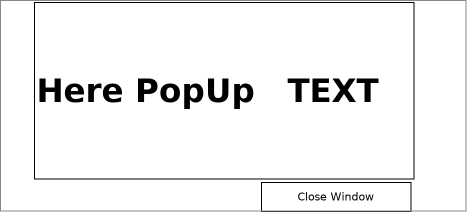
VISUALIZATION W01_PopupScreen  // 467x212
    Label (24,34 443x139)
    RoundedRectangle (261,182 150x30), "Close Window"
        OnMouseClick: CloseDialog Dialog=W01_PopupScreen, Result=OK, NumpadKeypadSet=True
    Rectangle (34,2 380x177), "Here PopUp TEXT"
END_VISUALIZATION

(* stored: Version 1.1.0.1, ProductVersion 3.1.4024.4
   Visu W01_PopupScreen: Id {a139f082-769d-4807-94eb-78ce2953c4c5} *)
